FUNCTION_BLOCK CylinderVtem IMPLEMENTS ICylinder
VAR
	vtem				: VtemByFesto;
END_VAR

;

METHOD bwd
vtem.moveBwd();
END_METHOD

METHOD fwd
vtem.moveFwd();
END_METHOD

END_FUNCTION_BLOCK

(* stored: Version 1.1.0.1, ProductVersion 3.1.4024.12
   POU CylinderVtem: Id {9c7ae81a-14b8-48a4-ac6a-92ee45d27ad6}, SpecialFunc None
   Method bwd: Id {485b6fd1-a845-4d7d-8395-dd9a39a8045d}
   Method fwd: Id {464facca-7b17-4e91-b35c-993bb7d4f533} *)
